FUNCTION_BLOCK PICKER_VIEW_NEW_BA (* View Composite FB *)
  (* Standard: 61499-2 *)
  (* Version 0.2, 2003-12-05, JHC, Rockwell Automation, Renamed from NEWCOMPFB. *)
  (* Version 0.1, 2002-01-08, JHC, Rockwell Automation, Added DLY FB as example. *)
  (* Version 0.0, 2000-05-27, JHC, Rockwell Automation *)
  (* Compiler header: package fb.rt.pnp;import fb.rt.vhmi.*;import fb.rt.math.*;import fb.rt.vmath.*; *)
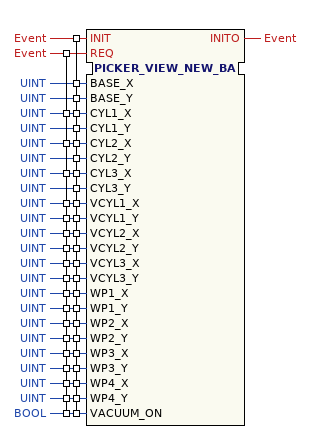
  EVENT_INPUT
    INIT WITH BASE_X, BASE_Y, CYL1_Y, CYL2_Y, CYL1_X, CYL2_X, VCYL1_X, VCYL1_Y, WP1_X, WP1_Y, VACUUM_ON, WP2_Y, WP2_X, WP3_X, WP3_Y, VCYL2_X, VCYL2_Y, VCYL3_X, VCYL3_Y, CYL3_X, CYL3_Y, WP4_X, WP4_Y; (* Initialization Request *)
    REQ WITH CYL1_X, CYL2_X, VCYL1_X, VCYL1_Y, WP1_X, WP1_Y, VACUUM_ON, WP2_X, WP2_Y, WP3_X, WP3_Y, CYL3_X, VCYL2_X, VCYL2_Y, VCYL3_X, VCYL3_Y, WP4_X, WP4_Y; (* Normal Execution Request *)
  END_EVENT
  EVENT_OUTPUT
    INITO; (* Initialization Confirm *)
  END_EVENT
  VAR_INPUT
    BASE_X : UINT;
    BASE_Y : UINT;
    CYL1_X : UINT;
    CYL1_Y : UINT;
    CYL2_X : UINT;
    CYL2_Y : UINT;
    CYL3_X : UINT;
    CYL3_Y : UINT;
    VCYL1_X : UINT;
    VCYL1_Y : UINT;
    VCYL2_X : UINT;
    VCYL2_Y : UINT;
    VCYL3_X : UINT;
    VCYL3_Y : UINT;
    WP1_X : UINT;
    WP1_Y : UINT;
    WP2_X : UINT;
    WP2_Y : UINT;
    WP3_X : UINT;
    WP3_Y : UINT;
    WP4_X : UINT;
    WP4_Y : UINT;
    VACUUM_ON : BOOL;
  END_VAR
  FBS
    PICKER_BASE : Render(name := "/fb/rt/pnp/picker_base_only.png", Display := 1, Layer := 13);
    PICKER_CYL1 : Render(name := "/fb/rt/pnp/cyl/cyl-1.png", Display := 1, Layer := 12);
    PICKER_CYL2 : Render(name := "/fb/rt/pnp/cyl/cyl-1.png", Display := 1, Layer := 11);
    PICKER_VCYL1 : Render(name := "/fb/rt/pnp/cyl/cylv-1.png", Display := 1, Layer := 9);
    WP1 : Render(name := "/fb/rt/pnp/workpiece.png", Display := 1, Layer := 14);
    PICKER_VACUUMON : Render(name := "/fb/rt/pnp/cyl/vacuum_on.png", Layer := 15);
    wp_place1 : Render(PosX := 534, PosY := 390, Display := 1, Layer := 1, name := "/fb/rt/pnp/wp_place.png");
    wp_place2 : Render(name := "/fb/rt/pnp/wp_place.png", PosX := 609, PosY := 540, Display := 1, Layer := 1);
    wp_place3 : Render(name := "/fb/rt/pnp/wp_place.png", PosX := 684, PosY := 465, Display := 1, Layer := 1);
    slider : Render(name := "/fb/rt/pnp/Slider.png", PosX := 459, PosY := 388, Display := 1, Layer := 1);
    WP2 : Render(name := "/fb/rt/pnp/workpiece1.png", Display := 1, Layer := 14);
    WP3 : Render(Display := 1, Layer := 14, name := "/fb/rt/pnp/workpiece2.png");
    PICKER_CYL3 : Render(name := "/fb/rt/pnp/cyl/cyl-2.png", Display := 1, Layer := 10);
    PICKER_VCYL2 : Render(name := "/fb/rt/pnp/cyl/cylv-1.png", Layer := 8, Display := 1);
    PICKER_VCYL3 : Render(name := "/fb/rt/pnp/cyl/cylv-1.png", Layer := 7, Display := 1);
    PICKER_PIS1 : Render(name := "/fb/rt/pnp/cyl/pis-1.png", Display := 1, Layer := 10);
    SHIFT_CYL1 : shift(Y2 := 0, X2 := 20);
    SHIFT_CYL2 : shift(X2 := 90, Y2 := 0);
    PICKER_PIS2 : Render(Layer := 9, Display := 1, name := "/fb/rt/pnp/cyl/pis-1.png");
    PICKER_PIS3 : Render(name := "/fb/rt/pnp/cyl/pis-2.png", Display := 1, Layer := 8);
    SHIFT_CYL3 : shift(X2 := 90, Y2 := 0);
    PICKER_VPIS1 : Render(name := "/fb/rt/pnp/cyl/pisv-1.png", Display := 1, Layer := 7);
    SHIFT_VCYL1 : shift(X2 := 180, Y2 := 0);
    PICKER_VPIS2 : Render(name := "/fb/rt/pnp/cyl/pisv-1.png", Display := 1, Layer := 6);
    SHIFT_VCYL2 : shift(X2 := 0, Y2 := 90);
    PICKER_VPIS3 : Render(name := "/fb/rt/pnp/cyl/pisv-1.png", Layer := 5, Display := 1);
    SHIFT_VCYL3 : shift(Y2 := 90, X2 := 0);
    SHIFT_VACUUM : shift(X2 := 0, Y2 := 80);
    PICKER_VACUUM : Render(name := "/fb/rt/pnp/cyl/vacuum.png", Display := 1, Layer := 10);
  END_FBS
  EVENT_CONNECTIONS
    INIT TO PICKER_BASE.INIT;
    PICKER_BASE.INITO TO PICKER_CYL1.INIT;
    REQ TO WP1.ChangeXY;
    REQ TO PICKER_VACUUMON.ChangeValidity;
    wp_place2.INITO TO wp_place3.INIT;
    WP1.INITO TO WP2.INIT;
    REQ TO WP2.ChangeXY;
    REQ TO WP3.ChangeXY;
    slider.INITO TO INITO;
    WP2.INITO TO WP3.INIT;
    wp_place1.INITO TO wp_place2.INIT;
    PICKER_CYL1.INITO TO PICKER_PIS1.INIT;
    REQ TO SHIFT_CYL1.REQ;
    SHIFT_CYL1.DONE TO PICKER_CYL1.ChangeXY;
    REQ TO PICKER_PIS1.ChangeXY;
    INIT TO SHIFT_CYL1.REQ;
    PICKER_CYL2.INITO TO PICKER_PIS2.INIT;
    REQ TO PICKER_PIS2.ChangeXY;
    PICKER_PIS1.INITO TO PICKER_CYL2.INIT;
    PICKER_PIS2.INITO TO PICKER_CYL3.INIT;
    INIT TO SHIFT_CYL2.REQ;
    SHIFT_CYL2.DONE TO PICKER_CYL2.ChangeXY;
    REQ TO SHIFT_CYL2.REQ;
    SHIFT_CYL3.DONE TO PICKER_CYL3.ChangeXY;
    INIT TO SHIFT_CYL3.REQ;
    REQ TO SHIFT_CYL3.REQ;
    PICKER_CYL3.INITO TO PICKER_PIS3.INIT;
    PICKER_PIS3.INITO TO PICKER_VCYL1.INIT;
    REQ TO PICKER_PIS3.ChangeXY;
    PICKER_VCYL1.INITO TO PICKER_VPIS1.INIT;
    PICKER_VCYL2.INITO TO PICKER_VPIS2.INIT;
    PICKER_VPIS2.INITO TO PICKER_VCYL3.INIT;
    PICKER_VCYL3.INITO TO PICKER_VPIS3.INIT;
    PICKER_VPIS3.INITO TO WP1.INIT;
    INIT TO SHIFT_VCYL1.REQ;
    REQ TO SHIFT_VCYL1.REQ;
    SHIFT_VCYL1.DONE TO PICKER_VCYL1.ChangeXY;
    REQ TO PICKER_VPIS1.ChangeXY;
    REQ TO PICKER_VPIS3.ChangeXY;
    REQ TO PICKER_VPIS2.ChangeXY;
    REQ TO SHIFT_VCYL3.REQ;
    INIT TO SHIFT_VCYL3.REQ;
    INIT TO SHIFT_VCYL2.REQ;
    REQ TO SHIFT_VCYL2.REQ;
    SHIFT_VCYL2.DONE TO PICKER_VCYL2.ChangeXY;
    SHIFT_VCYL3.DONE TO PICKER_VCYL3.ChangeXY;
    REQ TO SHIFT_VACUUM.REQ;
    INIT TO SHIFT_VACUUM.REQ;
    PICKER_VPIS1.INITO TO PICKER_VCYL2.INIT;
    PICKER_VACUUMON.INITO TO PICKER_VACUUM.INIT;
    PICKER_VACUUM.INITO TO wp_place1.INIT;
    SHIFT_VACUUM.DONE TO PICKER_VACUUM.ChangeXY;
    SHIFT_VACUUM.DONE TO PICKER_VACUUMON.ChangeXY;
    wp_place3.INITO TO slider.INIT;
    WP3.INITO TO PICKER_VACUUMON.INIT;
  END_CONNECTIONS
  DATA_CONNECTIONS
    VACUUM_ON TO PICKER_VACUUMON.Display;
    BASE_X TO PICKER_BASE.PosX;
    BASE_Y TO PICKER_BASE.PosY;
    WP1_X TO WP1.PosX;
    WP1_Y TO WP1.PosY;
    WP2_X TO WP2.PosX;
    WP2_Y TO WP2.PosY;
    WP3_X TO WP3.PosX;
    WP3_Y TO WP3.PosY;
    BASE_X TO SHIFT_CYL1.X1;
    SHIFT_CYL1.X TO PICKER_CYL1.PosX;
    SHIFT_CYL1.Y TO PICKER_CYL1.PosY;
    CYL1_X TO PICKER_PIS1.PosX;
    CYL1_Y TO PICKER_PIS1.PosY;
    BASE_Y TO SHIFT_CYL1.Y1;
    CYL2_X TO PICKER_PIS2.PosX;
    CYL2_Y TO PICKER_PIS2.PosY;
    CYL1_X TO SHIFT_CYL2.X1;
    CYL1_Y TO SHIFT_CYL2.Y1;
    SHIFT_CYL2.X TO PICKER_CYL2.PosX;
    SHIFT_CYL2.Y TO PICKER_CYL2.PosY;
    CYL2_X TO SHIFT_CYL3.X1;
    SHIFT_CYL3.X TO PICKER_CYL3.PosX;
    SHIFT_CYL3.Y TO PICKER_CYL3.PosY;
    CYL3_X TO PICKER_PIS3.PosX;
    CYL3_Y TO PICKER_PIS3.PosY;
    CYL2_Y TO SHIFT_CYL3.Y1;
    CYL3_X TO SHIFT_VCYL1.X1;
    CYL3_Y TO SHIFT_VCYL1.Y1;
    SHIFT_VCYL1.X TO PICKER_VCYL1.PosX;
    SHIFT_VCYL1.Y TO PICKER_VCYL1.PosY;
    VCYL1_X TO SHIFT_VCYL2.X1;
    VCYL1_Y TO SHIFT_VCYL2.Y1;
    VCYL2_Y TO SHIFT_VCYL3.Y1;
    VCYL2_X TO SHIFT_VCYL3.X1;
    SHIFT_VCYL2.X TO PICKER_VCYL2.PosX;
    SHIFT_VCYL2.Y TO PICKER_VCYL2.PosY;
    VCYL2_X TO PICKER_VPIS2.PosX;
    VCYL2_Y TO PICKER_VPIS2.PosY;
    VCYL3_X TO PICKER_VPIS3.PosX;
    VCYL3_Y TO PICKER_VPIS3.PosY;
    SHIFT_VCYL3.X TO PICKER_VCYL3.PosX;
    SHIFT_VCYL3.Y TO PICKER_VCYL3.PosY;
    VCYL1_X TO PICKER_VPIS1.PosX;
    VCYL1_Y TO PICKER_VPIS1.PosY;
    VCYL3_X TO SHIFT_VACUUM.X1;
    VCYL3_Y TO SHIFT_VACUUM.Y1;
    SHIFT_VACUUM.X TO PICKER_VACUUM.PosX;
    SHIFT_VACUUM.Y TO PICKER_VACUUM.PosY;
    SHIFT_VACUUM.X TO PICKER_VACUUMON.PosX;
    SHIFT_VACUUM.Y TO PICKER_VACUUMON.PosY;
  END_CONNECTIONS
END_FUNCTION_BLOCK
